PROGRAM MAIN
VAR
	a: DWORD;
END_VAR

//a:=a+1;
//1

END_PROGRAM

(* stored: Version 1.1.0.1, ProductVersion 3.1.4024.10
   POU MAIN: Id {a3057a8d-5e3c-4200-b437-c3c219daaac9}, SpecialFunc None *)
